{attribute 'qualified_only'}
{attribute 'strict'}
{attribute 'to_string'}
TYPE E_EM_InfeedConveyor_Seq_Execute :
(
	Idle := c_nSeqIdle,
	Start := c_nSeqStart,
	
	WaitForProduct,
	
	MoveProductToDoor, 
	WaitUntilLiftReady,
	RequestLiftReceiving,
	OpenDoor,
	MoveProductInLift,
	CloseDoor,
	
	
	
	Ready := c_nSeqReady,
	Error := c_nSeqError

);
END_TYPE

(* stored: Version 1.1.0.1, ProductVersion 3.1.4026.13
   DUT E_EM_InfeedConveyor_Seq_Execute: Id {e602f4c8-8aa5-4c18-9cfc-cb41bfdf5cfd} *)
